RoboDK station: Sheet C - Bottom.rdk

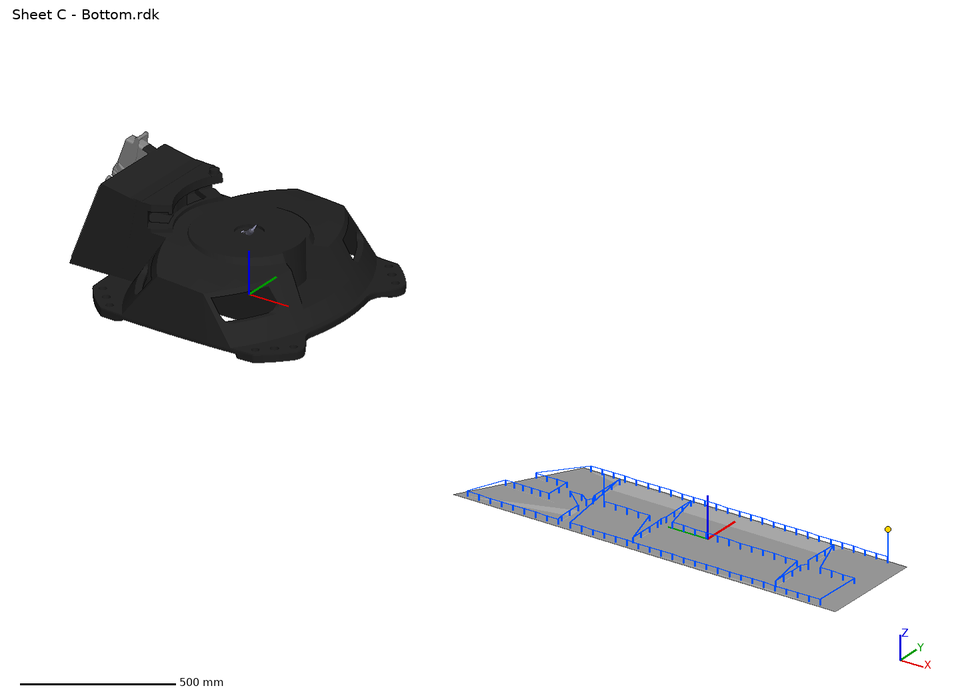
[picture v0: the station drawn from its stored meshes, robots at their saved joint values, targets as dots, program paths as lines]
Station Sheet C - Bottom (saved by RoboDK 5.2.3). Poses are relative to the parent item; angles as X-Y-Z fixed-axis rotations.
  - frame KUKA KR 210 R2700 extra Base at (0, 0, 0) mm
    - robot KUKA KR 210 R2700 extra: 6 axes, payload 210 kg, reach 2696 mm, repeatability 0.06 mm, weight 1068 kg
        joint limits [-185, -140, -120, -350, -125, -350] to [185, -5, 155, 350, 125, 350]; home [0, -90, 90, 0, 0, 0]; saved at [0.009, -34.349, 130.969, 180.008, 45.62, -179.999]
      - tool Spindle, TCP at (32, 0, 260) mm, rotated rx 0 ry 39 rz 0 deg, size 157.3 x 72 x 259.9 mm
  - frame Frame 2 at (1800, 0, -372.68) mm, rotated rx 0 ry 0 rz 90 deg
    - object Box 1 - Sheet C -  Bottom at (0, 0, 0) mm, size 400 x 1500 x 0.8 mm, geometry from Box 1 - Sheet C -  Bottom.stl
    - object Sheet C-box 1 Hole positioning Bottom at (0, 0, 0) mm, 120 curves, geometry from Point 120
  - machining project Path1 settings: rotZ(0) | rotX(0)*rotY(0) | rotz(0) | onStart | onPathStart | onApproach | onPoint | onRetract | onFinish | SetRPM(%1) | SetTool(%1) | Extruder(%1) | default | default | OutOnMov(%1) | OutOffMov(%1) | onPathFinish | M_RunCode(%1)
  - program Path1 (611 instructions, listed below)
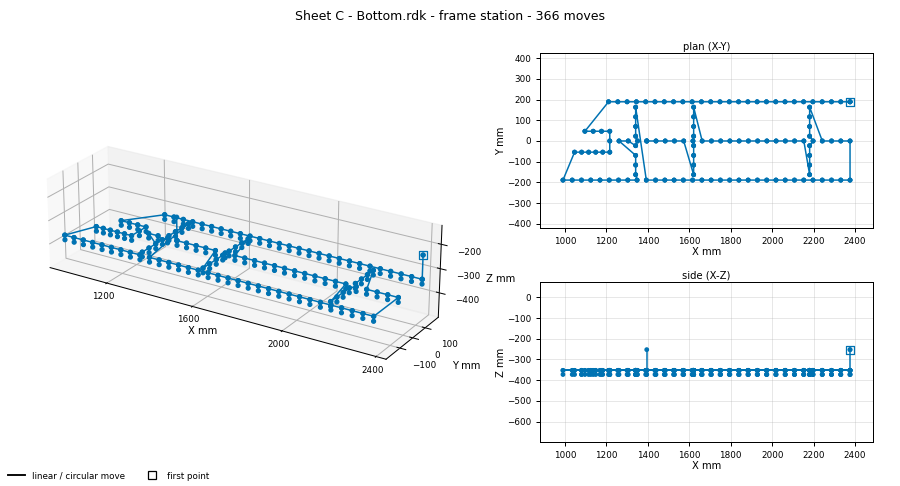
[picture p0: tool path of Sheet C - Bottom.rdk in frame station, 366 of 366 moves have a stored position in this frame; points joined in program order, loops and branches not executed]

--- program Path1 (robot KUKA KR 210 R2700 extra) ---
  Smooth(1)
  Set speed (1000.0 mm/s)
  Set Ref.: Frame 2
  Set Tool: Spindle
  Show Spindle
  MoveJ 1 to (189, -575.99, 120) mm, rotated rx -180 ry 0 rz 90 deg; joints [-5.138, -22.439, 74.968, 113.656, 3.528, -117.694]
  MoveL 2 to (189, -575.99, 120) mm, rotated rx -180 ry 0 rz 90 deg; joints [-5.138, -22.439, 74.968, 113.656, 3.528, -117.694]
  MoveL 3 to (189, -575.99, 20) mm, rotated rx 180 ry 0 rz 90 deg; joints [-5.138, -18.208, 72.448, 134.025, 4.496, -138.111]
  MoveL 4 to (189, -575.99, 20) mm, rotated rx 180 ry 0 rz 90 deg; joints [-5.138, -18.208, 72.448, 134.025, 4.496, -138.111]
  Set speed (50.0 mm/s)
  MoveL 5 to (189, -575.99, 0) mm, rotated rx -180 ry 0 rz 90 deg; joints [-5.138, -17.345, 71.889, 136.67, 4.711, -140.764]
  MoveL 6 to (189, -575.99, 20) mm, rotated rx 180 ry 0 rz 90 deg; joints [-5.138, -18.208, 72.448, 134.025, 4.496, -138.111]
  Set speed (1000.0 mm/s)
  MoveL 7 to (189, -531.14, 20) mm, rotated rx -180 ry 0 rz 90 deg; joints [-5.249, -19.449, 75.768, 147.536, 6.158, -151.77]
  Set speed (50.0 mm/s)
  MoveL 8 to (189, -531.14, 0) mm, rotated rx 180 ry 0 rz 90 deg; joints [-5.249, -18.579, 75.216, 149.054, 6.429, -153.297]
  MoveL 9 to (189, -531.14, 20) mm, rotated rx -180 ry 0 rz 90 deg; joints [-5.249, -19.449, 75.768, 147.536, 6.158, -151.77]
  Set speed (1000.0 mm/s)
  MoveL 10 to (189, -486.3, 20) mm, rotated rx 180 ry 0 rz 90 deg; joints [-5.366, -20.604, 78.961, 154.91, 7.977, -159.298]
  Set speed (50.0 mm/s)
  MoveL 11 to (189, -486.3, 0) mm, rotated rx -180 ry 0 rz 90 deg; joints [-5.366, -19.726, 78.415, 155.882, 8.281, -160.28]
  MoveL 12 to (189, -486.3, 20) mm, rotated rx 180 ry 0 rz 90 deg; joints [-5.366, -20.604, 78.961, 154.91, 7.977, -159.298]
  Set speed (1000.0 mm/s)
  MoveL 13 to (189, -441.45, 20) mm, rotated rx -180 ry 0 rz 90 deg; joints [-5.487, -21.682, 82.042, 159.405, 9.85, -163.953]
  Set speed (50.0 mm/s)
  MoveL 14 to (189, -441.45, 0) mm, rotated rx 180 ry 0 rz 90 deg; joints [-5.487, -20.792, 81.501, 160.086, 10.177, -164.645]
  MoveL 15 to (189, -441.45, 20) mm, rotated rx -180 ry 0 rz 90 deg; joints [-5.487, -21.682, 82.042, 159.405, 9.85, -163.953]
  Set speed (1000.0 mm/s)
  MoveL 16 to (189, -396.61, 20) mm, rotated rx 180 ry 0 rz 90 deg; joints [-5.615, -22.684, 85.023, 162.387, 11.74, -167.102]
  Set speed (50.0 mm/s)
  MoveL 17 to (189, -396.61, 0) mm, rotated rx 180 ry 0 rz 90 deg; joints [-5.615, -21.783, 84.484, 162.898, 12.086, -167.625]
  MoveL 18 to (189, -396.61, 20) mm, rotated rx 180 ry 0 rz 90 deg; joints [-5.615, -22.684, 85.023, 162.387, 11.74, -167.102]
  Set speed (1000.0 mm/s)
  MoveL 19 to (189, -351.76, 20) mm, rotated rx 180 ry 0 rz 90 deg; joints [-5.748, -23.614, 87.912, 164.494, 13.636, -169.383]
  Set speed (50.0 mm/s)
  MoveL 20 to (189, -351.76, 0) mm, rotated rx -180 ry 0 rz 90 deg; joints [-5.748, -22.7, 87.374, 164.896, 13.998, -169.798]
  MoveL 21 to (189, -351.76, 20) mm, rotated rx 180 ry 0 rz 90 deg; joints [-5.748, -23.614, 87.912, 164.494, 13.636, -169.383]
  Set speed (1000.0 mm/s)
  MoveL 22 to (189, -306.91, 20) mm, rotated rx 180 ry 0 rz 90 deg; joints [-5.887, -24.475, 90.718, 166.05, 15.532, -171.123]
  Set speed (50.0 mm/s)
  MoveL 23 to (189, -306.91, 0) mm, rotated rx 180 ry 0 rz 90 deg; joints [-5.887, -23.547, 90.179, 166.379, 15.909, -171.464]
  MoveL 24 to (189, -306.91, 20) mm, rotated rx 180 ry 0 rz 90 deg; joints [-5.887, -24.475, 90.718, 166.05, 15.532, -171.123]
  Set speed (1000.0 mm/s)
  MoveL 25 to (189, -262.07, 20) mm, rotated rx 180 ry 0 rz 90 deg; joints [-6.034, -25.267, 93.445, 167.24, 17.428, -172.504]
  Set speed (50.0 mm/s)
  MoveL 26 to (189, -262.07, 0) mm, rotated rx 180 ry 0 rz 90 deg; joints [-6.034, -24.325, 92.905, 167.516, 17.821, -172.794]
  MoveL 27 to (189, -262.07, 20) mm, rotated rx 180 ry 0 rz 90 deg; joints [-6.034, -25.267, 93.445, 167.24, 17.428, -172.504]
  Set speed (1000.0 mm/s)
  MoveL 28 to (189, -217.22, 20) mm, rotated rx 180 ry 0 rz 90 deg; joints [-6.188, -25.991, 96.102, 168.173, 19.328, -173.639]
  Set speed (50.0 mm/s)
  MoveL 29 to (189, -217.22, 0) mm, rotated rx 180 ry 0 rz 90 deg; joints [-6.188, -25.033, 95.559, 168.41, 19.734, -173.891]
  MoveL 30 to (189, -217.22, 20) mm, rotated rx 180 ry 0 rz 90 deg; joints [-6.188, -25.991, 96.102, 168.173, 19.328, -173.639]
  Set speed (1000.0 mm/s)
  MoveL 31 to (189, -172.37, 20) mm, rotated rx -180 ry 0 rz 90 deg; joints [-6.35, -26.648, 98.692, 168.919, 21.233, -174.597]
  Set speed (50.0 mm/s)
  MoveL 32 to (189, -172.37, 0) mm, rotated rx -180 ry 0 rz 90 deg; joints [-6.35, -25.673, 98.145, 169.126, 21.652, -174.82]
  MoveL 33 to (189, -172.37, 20) mm, rotated rx -180 ry 0 rz 90 deg; joints [-6.35, -26.648, 98.692, 168.919, 21.233, -174.597]
  Set speed (1000.0 mm/s)
  MoveL 34 to (189, -127.53, 20) mm, rotated rx -180 ry 0 rz 90 deg; joints [-6.521, -27.237, 101.217, 169.524, 23.145, -175.427]
  Set speed (50.0 mm/s)
  MoveL 35 to (189, -127.53, 0) mm, rotated rx -180 ry 0 rz 90 deg; joints [-6.521, -26.244, 100.665, 169.708, 23.578, -175.627]
  MoveL 36 to (189, -127.53, 20) mm, rotated rx -180 ry 0 rz 90 deg; joints [-6.521, -27.237, 101.217, 169.524, 23.145, -175.427]
  Set speed (1000.0 mm/s)
  MoveL 37 to (189, -82.68, 20) mm, rotated rx 180 ry 0 rz 90 deg; joints [-6.701, -27.756, 103.683, 170.02, 25.07, -176.161]
  Set speed (50.0 mm/s)
  MoveL 38 to (189, -82.68, 0) mm, rotated rx 180 ry 0 rz 90 deg; joints [-6.701, -26.744, 103.125, 170.184, 25.516, -176.343]
  MoveL 39 to (189, -82.68, 20) mm, rotated rx 180 ry 0 rz 90 deg; joints [-6.701, -27.756, 103.683, 170.02, 25.07, -176.161]
  Set speed (1000.0 mm/s)
  MoveL 40 to (189, -37.84, 20) mm, rotated rx -180 ry 0 rz 90 deg; joints [-6.891, -28.203, 106.092, 170.429, 27.009, -176.822]
  Set speed (50.0 mm/s)
  MoveL 41 to (189, -37.84, 0) mm, rotated rx -180 ry 0 rz 90 deg; joints [-6.891, -27.173, 105.527, 170.578, 27.468, -176.99]
  MoveL 42 to (189, -37.84, 20) mm, rotated rx -180 ry 0 rz 90 deg; joints [-6.891, -28.203, 106.092, 170.429, 27.009, -176.822]
  Set speed (1000.0 mm/s)
  MoveL 43 to (189, 7.01, 20) mm, rotated rx 180 ry 0 rz 90 deg; joints [-7.093, -28.577, 108.445, 170.767, 28.968, -177.429]
  Set speed (50.0 mm/s)
  MoveL 44 to (189, 7.01, 0) mm, rotated rx -180 ry 0 rz 90 deg; joints [-7.093, -27.526, 107.872, 170.903, 29.44, -177.585]
  MoveL 45 to (189, 7.01, 20) mm, rotated rx 180 ry 0 rz 90 deg; joints [-7.093, -28.577, 108.445, 170.767, 28.968, -177.429]
  Set speed (1000.0 mm/s)
  MoveL 46 to (189, 51.86, 20) mm, rotated rx -180 ry 0 rz 90 deg; joints [-7.306, -28.875, 110.745, 171.047, 30.95, -177.996]
  Set speed (50.0 mm/s)
  MoveL 47 to (189, 51.86, 0) mm, rotated rx 180 ry 0 rz 90 deg; joints [-7.306, -27.803, 110.163, 171.172, 31.434, -178.142]
  MoveL 48 to (189, 51.86, 20) mm, rotated rx -180 ry 0 rz 90 deg; joints [-7.306, -28.875, 110.745, 171.047, 30.95, -177.996]
  Set speed (1000.0 mm/s)
  MoveL 49 to (189, 96.7, 20) mm, rotated rx 180 ry 0 rz 90 deg; joints [-7.533, -29.093, 112.992, 171.278, 32.96, -178.532]
  Set speed (50.0 mm/s)
  MoveL 50 to (189, 96.7, 0) mm, rotated rx 180 ry 0 rz 90 deg; joints [-7.533, -27.999, 112.4, 171.393, 33.456, -178.67]
  MoveL 51 to (189, 96.7, 20) mm, rotated rx 180 ry 0 rz 90 deg; joints [-7.533, -29.093, 112.992, 171.278, 32.96, -178.532]
  Set speed (1000.0 mm/s)
  MoveL 52 to (189, 141.55, 20) mm, rotated rx 180 ry 0 rz 90 deg; joints [-7.774, -29.227, 115.187, 171.465, 35.001, -179.048]
  Set speed (50.0 mm/s)
  MoveL 53 to (189, 141.55, 0) mm, rotated rx -180 ry 0 rz 90 deg; joints [-7.774, -28.111, 114.584, 171.572, 35.509, -179.179]
  MoveL 54 to (189, 141.55, 20) mm, rotated rx 180 ry 0 rz 90 deg; joints [-7.774, -29.227, 115.187, 171.465, 35.001, -179.048]
  Set speed (1000.0 mm/s)
  MoveL 55 to (189, 186.39, 20) mm, rotated rx -180 ry 0 rz 90 deg; joints [-8.031, -29.272, 117.331, 171.615, 37.079, -179.55]
  Set speed (50.0 mm/s)
  MoveL 56 to (189, 186.39, 0) mm, rotated rx 180 ry 0 rz 90 deg; joints [-8.031, -28.133, 116.716, 171.714, 37.597, -179.676]
  MoveL 57 to (189, 186.39, 20) mm, rotated rx -180 ry 0 rz 90 deg; joints [-8.031, -29.272, 117.331, 171.615, 37.079, -179.55]
  Set speed (1000.0 mm/s)
  MoveL 58 to (189, 231.24, 20) mm, rotated rx -180 ry 0 rz 90 deg; joints [-8.305, -29.223, 119.424, 171.73, 39.199, -180.046]
  Set speed (50.0 mm/s)
  MoveL 59 to (189, 231.24, 0) mm, rotated rx 180 ry 0 rz 90 deg; joints [-8.305, -28.061, 118.796, 171.823, 39.727, -180.166]
  MoveL 60 to (189, 231.24, 20) mm, rotated rx -180 ry 0 rz 90 deg; joints [-8.305, -29.223, 119.424, 171.73, 39.199, -180.046]
  Set speed (1000.0 mm/s)
  MoveL 61 to (189, 276.09, 20) mm, rotated rx -180 ry 0 rz 90 deg; joints [-8.599, -29.075, 121.466, 171.814, 41.365, -180.541]
  Set speed (50.0 mm/s)
  MoveL 62 to (189, 276.09, 0) mm, rotated rx -180 ry 0 rz 90 deg; joints [-8.599, -27.889, 120.823, 171.901, 41.903, -180.657]
  MoveL 63 to (189, 276.09, 20) mm, rotated rx -180 ry 0 rz 90 deg; joints [-8.599, -29.075, 121.466, 171.814, 41.365, -180.541]
  Set speed (1000.0 mm/s)
  MoveL 64 to (189, 320.93, 20) mm, rotated rx 180 ry 0 rz 90 deg; joints [-8.914, -28.82, 123.454, 171.868, 43.583, -181.04]
  Set speed (50.0 mm/s)
  MoveL 65 to (189, 320.93, 0) mm, rotated rx -180 ry 0 rz 90 deg; joints [-8.914, -27.611, 122.796, 171.949, 44.129, -181.153]
  MoveL 66 to (189, 320.93, 20) mm, rotated rx 180 ry 0 rz 90 deg; joints [-8.914, -28.82, 123.454, 171.868, 43.583, -181.04]
  Set speed (1000.0 mm/s)
  MoveL 67 to (189, 365.78, 20) mm, rotated rx 180 ry 0 rz 90 deg; joints [-9.253, -28.451, 125.389, 171.894, 45.859, -181.551]
  Set speed (50.0 mm/s)
  MoveL 68 to (189, 365.78, 0) mm, rotated rx -180 ry 0 rz 90 deg; joints [-9.253, -27.219, 124.715, 171.969, 46.412, -181.66]
  MoveL 69 to (189, 365.78, 20) mm, rotated rx 180 ry 0 rz 90 deg; joints [-9.253, -28.451, 125.389, 171.894, 45.859, -181.551]
  Set speed (1000.0 mm/s)
  MoveL 70 to (189, 410.63, 20) mm, rotated rx 180 ry 0 rz 90 deg; joints [-9.618, -27.959, 127.268, 171.892, 48.199, -182.078]
  Set speed (50.0 mm/s)
  MoveL 71 to (189, 410.63, 0) mm, rotated rx 180 ry 0 rz 90 deg; joints [-9.618, -26.705, 126.576, 171.962, 48.756, -182.183]
  MoveL 72 to (189, 410.63, 20) mm, rotated rx 180 ry 0 rz 90 deg; joints [-9.618, -27.959, 127.268, 171.892, 48.199, -182.078]
  Set speed (1000.0 mm/s)
  MoveL 73 to (189, 455.47, 20) mm, rotated rx -180 ry 0 rz 90 deg; joints [-10.013, -27.337, 129.088, 171.86, 50.607, -182.626]
  Set speed (50.0 mm/s)
  MoveL 74 to (189, 455.47, 0) mm, rotated rx 180 ry 0 rz 90 deg; joints [-10.013, -26.061, 128.379, 171.925, 51.167, -182.729]
  MoveL 75 to (189, 455.47, 20) mm, rotated rx -180 ry 0 rz 90 deg; joints [-10.013, -27.337, 129.088, 171.86, 50.607, -182.626]
  Set speed (1000.0 mm/s)
  MoveL 76 to (189, 500.32, 20) mm, rotated rx -180 ry 0 rz 90 deg; joints [-10.441, -26.573, 130.848, 171.8, 53.091, -183.204]
  Set speed (50.0 mm/s)
  MoveL 77 to (189, 500.32, 0) mm, rotated rx 180 ry 0 rz 90 deg; joints [-10.441, -25.278, 130.119, 171.859, 53.651, -183.304]
  MoveL 78 to (189, 500.32, 20) mm, rotated rx -180 ry 0 rz 90 deg; joints [-10.441, -26.573, 130.848, 171.8, 53.091, -183.204]
  Set speed (1000.0 mm/s)
  MoveL 79 to (189, 545.16, 20) mm, rotated rx 180 ry 0 rz 90 deg; joints [-10.907, -25.659, 132.544, 171.708, 55.656, -183.817]
  Set speed (50.0 mm/s)
  MoveL 80 to (189, 545.16, 0) mm, rotated rx -180 ry 0 rz 90 deg; joints [-10.907, -24.347, 131.794, 171.762, 56.212, -183.914]
  MoveL 81 to (189, 545.16, 20) mm, rotated rx 180 ry 0 rz 90 deg; joints [-10.907, -25.659, 132.544, 171.708, 55.656, -183.817]
  Set speed (1000.0 mm/s)
  MoveL 82 to (189, 590.01, 20) mm, rotated rx 180 ry 0 rz 90 deg; joints [-11.417, -24.583, 134.171, 171.582, 58.308, -184.473]
  Set speed (50.0 mm/s)
  MoveL 83 to (189, 590.01, 0) mm, rotated rx 180 ry 0 rz 90 deg; joints [-11.417, -23.257, 133.4, 171.631, 58.856, -184.568]
  MoveL 84 to (189, 590.01, 20) mm, rotated rx 180 ry 0 rz 90 deg; joints [-11.417, -24.583, 134.171, 171.582, 58.308, -184.473]
  Set speed (1000.0 mm/s)
  MoveL 85 to (46.83, 704.01, 20) mm, rotated rx -180 ry 0 rz 90 deg; joints [-3.261, -20.272, 138.599, 177.776, 67.298, -181.677]
  Set speed (50.0 mm/s)
  MoveL 86 to (46.83, 704.01, 0) mm, rotated rx -180 ry 0 rz 90 deg; joints [-3.261, -18.933, 137.76, 177.784, 67.797, -181.698]
  MoveL 87 to (46.83, 704.01, 20) mm, rotated rx -180 ry 0 rz 90 deg; joints [-3.261, -20.272, 138.599, 177.776, 67.298, -181.677]
  Set speed (1000.0 mm/s)
  MoveL 88 to (46.83, 664.01, 20) mm, rotated rx -180 ry 0 rz 90 deg; joints [-3.11, -21.766, 137.33, 177.833, 64.539, -181.486]
  Set speed (50.0 mm/s)
  MoveL 89 to (46.83, 664.01, 0) mm, rotated rx 180 ry 0 rz 90 deg; joints [-3.11, -20.425, 136.512, 177.842, 65.061, -181.508]
  MoveL 90 to (46.83, 664.01, 20) mm, rotated rx -180 ry 0 rz 90 deg; joints [-3.11, -21.766, 137.33, 177.833, 64.539, -181.486]
  Set speed (1000.0 mm/s)
  MoveL 91 to (46.83, 624.01, 20) mm, rotated rx -180 ry 0 rz 90 deg; joints [-2.972, -23.094, 135.993, 177.88, 61.877, -181.311]
  Set speed (50.0 mm/s)
  MoveL 92 to (46.83, 624.01, 0) mm, rotated rx -180 ry 0 rz 90 deg; joints [-2.972, -21.757, 135.196, 177.89, 62.416, -181.333]
  MoveL 93 to (46.83, 624.01, 20) mm, rotated rx -180 ry 0 rz 90 deg; joints [-2.972, -23.094, 135.993, 177.88, 61.877, -181.311]
  Set speed (1000.0 mm/s)
  MoveL 94 to (46.83, 584.01, 20) mm, rotated rx -180 ry 0 rz 90 deg; joints [-2.846, -24.267, 134.593, 177.917, 59.309, -181.149]
  Set speed (50.0 mm/s)
  MoveL 95 to (46.83, 584.01, 0) mm, rotated rx 180 ry 0 rz 90 deg; joints [-2.846, -22.938, 133.816, 177.929, 59.86, -181.173]
  MoveL 96 to (46.83, 584.01, 20) mm, rotated rx -180 ry 0 rz 90 deg; joints [-2.846, -24.267, 134.593, 177.917, 59.309, -181.149]
  Set speed (1000.0 mm/s)
  MoveL 97 to (-0.17, 584.01, 20) mm, rotated rx -180 ry 0 rz 90 deg; joints [0.01, -24.235, 134.635, 180.008, 59.4, -179.996]
  Set speed (50.0 mm/s)
  MoveL 98 to (-0.17, 584.01, 0) mm, rotated rx -180 ry 0 rz 90 deg; joints [0.01, -22.906, 133.857, 180.008, 59.952, -179.996]
  MoveL 99 to (-0.17, 584.01, 20) mm, rotated rx -180 ry 0 rz 90 deg; joints [0.01, -24.235, 134.635, 180.008, 59.4, -179.996]
  Set speed (1000.0 mm/s)
  MoveL 100 to (-54.17, 584.01, 20) mm, rotated rx -180 ry 0 rz 90 deg; joints [3.291, -24.277, 134.579, 182.409, 59.278, -178.672]
  Set speed (50.0 mm/s)
  MoveL 101 to (-54.17, 584.01, 0) mm, rotated rx 180 ry 0 rz 90 deg; joints [3.291, -22.949, 133.803, 182.395, 59.829, -178.645]
  MoveL 102 to (-54.17, 584.01, 20) mm, rotated rx -180 ry 0 rz 90 deg; joints [3.291, -24.277, 134.579, 182.409, 59.278, -178.672]
  Set speed (1000.0 mm/s)
  MoveL 103 to (-54.17, 618.01, 20) mm, rotated rx -180 ry 0 rz 90 deg; joints [3.414, -23.292, 135.773, 182.445, 61.453, -178.514]
  Set speed (50.0 mm/s)
  MoveL 104 to (-54.17, 618.01, 0) mm, rotated rx 180 ry 0 rz 90 deg; joints [3.414, -21.957, 134.979, 182.433, 61.994, -178.488]
  MoveL 105 to (-54.17, 618.01, 20) mm, rotated rx -180 ry 0 rz 90 deg; joints [3.414, -23.292, 135.773, 182.445, 61.453, -178.514]
  Set speed (1000.0 mm/s)
  MoveL 106 to (-54.17, 652.01, 20) mm, rotated rx -180 ry 0 rz 90 deg; joints [3.547, -22.196, 136.922, 182.489, 63.694, -178.346]
  Set speed (50.0 mm/s)
  MoveL 107 to (-54.17, 652.01, 0) mm, rotated rx -180 ry 0 rz 90 deg; joints [3.547, -20.856, 136.11, 182.478, 64.221, -178.32]
  MoveL 108 to (-54.17, 652.01, 20) mm, rotated rx -180 ry 0 rz 90 deg; joints [3.547, -22.196, 136.922, 182.489, 63.694, -178.346]
  Set speed (1000.0 mm/s)
  MoveL 109 to (-54.17, 686.01, 20) mm, rotated rx -180 ry 0 rz 90 deg; joints [3.69, -20.982, 138.023, 182.541, 66.004, -178.165]
  Set speed (50.0 mm/s)
  MoveL 110 to (-54.17, 686.01, 0) mm, rotated rx -180 ry 0 rz 90 deg; joints [3.69, -19.641, 137.193, 182.531, 66.514, -178.14]
  MoveL 111 to (-54.17, 686.01, 20) mm, rotated rx -180 ry 0 rz 90 deg; joints [3.69, -20.982, 138.023, 182.541, 66.004, -178.165]
  Set speed (1000.0 mm/s)
  MoveL 112 to (-54.17, 720.01, 20) mm, rotated rx -180 ry 0 rz 90 deg; joints [3.845, -19.645, 139.073, 182.602, 68.386, -177.969]
  Set speed (50.0 mm/s)
  MoveL 113 to (-54.17, 720.01, 0) mm, rotated rx 180 ry 0 rz 90 deg; joints [3.845, -18.308, 138.226, 182.593, 68.874, -177.945]
  MoveL 114 to (-54.17, 720.01, 20) mm, rotated rx -180 ry 0 rz 90 deg; joints [3.845, -19.645, 139.073, 182.602, 68.386, -177.969]
  Set speed (1000.0 mm/s)
  MoveL 115 to (-54.17, 754.01, 20) mm, rotated rx 180 ry 0 rz 90 deg; joints [4.014, -18.181, 140.071, 182.673, 70.84, -177.756]
  Set speed (50.0 mm/s)
  MoveL 116 to (-54.17, 754.01, 0) mm, rotated rx -180 ry 0 rz 90 deg; joints [4.014, -16.852, 139.205, 182.666, 71.302, -177.734]
  MoveL 117 to (-54.17, 754.01, 20) mm, rotated rx 180 ry 0 rz 90 deg; joints [4.014, -18.181, 140.071, 182.673, 70.84, -177.756]
  Set speed (1000.0 mm/s)
  MoveL 118 to (-189, 810.01, 20) mm, rotated rx 180 ry 0 rz 90 deg; joints [14.788, -16.611, 140.997, 189.687, 72.681, -171.315]
  Set speed (50.0 mm/s)
  MoveL 119 to (-189, 810.01, 0) mm, rotated rx 180 ry 0 rz 90 deg; joints [14.788, -15.296, 140.112, 189.664, 73.105, -171.239]
  MoveL 120 to (-189, 810.01, 20) mm, rotated rx 180 ry 0 rz 90 deg; joints [14.788, -16.611, 140.997, 189.687, 72.681, -171.315]
  Set speed (1000.0 mm/s)
  MoveL 121 to (-189, 765.3, 20) mm, rotated rx -180 ry 0 rz 90 deg; joints [13.954, -18.623, 139.784, 189.319, 69.574, -172.348]
  Set speed (50.0 mm/s)
  MoveL 122 to (-189, 765.3, 0) mm, rotated rx -180 ry 0 rz 90 deg; joints [13.954, -17.292, 138.923, 189.291, 70.039, -172.267]
  MoveL 123 to (-189, 765.3, 20) mm, rotated rx -180 ry 0 rz 90 deg; joints [13.954, -18.623, 139.784, 189.319, 69.574, -172.348]
  Set speed (1000.0 mm/s)
  MoveL 124 to (-189, 720.59, 20) mm, rotated rx 180 ry 0 rz 90 deg; joints [13.207, -20.428, 138.476, 189.016, 66.561, -173.276]
  Set speed (50.0 mm/s)
  MoveL 125 to (-189, 720.59, 0) mm, rotated rx -180 ry 0 rz 90 deg; joints [13.207, -19.088, 137.639, 188.983, 67.057, -173.19]
  MoveL 126 to (-189, 720.59, 20) mm, rotated rx 180 ry 0 rz 90 deg; joints [13.207, -20.428, 138.476, 189.016, 66.561, -173.276]
  Set speed (1000.0 mm/s)
  MoveL 127 to (-189, 675.88, 20) mm, rotated rx -180 ry 0 rz 90 deg; joints [12.535, -22.031, 137.08, 188.768, 63.643, -174.114]
  Set speed (50.0 mm/s)
  MoveL 128 to (-189, 675.88, 0) mm, rotated rx 180 ry 0 rz 90 deg; joints [12.535, -20.691, 136.266, 188.729, 64.163, -174.025]
  MoveL 129 to (-189, 675.88, 20) mm, rotated rx -180 ry 0 rz 90 deg; joints [12.535, -22.031, 137.08, 188.768, 63.643, -174.114]
  Set speed (1000.0 mm/s)
  MoveL 130 to (-189, 631.17, 20) mm, rotated rx 180 ry 0 rz 90 deg; joints [11.927, -23.443, 135.601, 188.567, 60.822, -174.878]
  Set speed (50.0 mm/s)
  MoveL 131 to (-189, 631.17, 0) mm, rotated rx -180 ry 0 rz 90 deg; joints [11.927, -22.109, 134.809, 188.522, 61.359, -174.786]
  MoveL 132 to (-189, 631.17, 20) mm, rotated rx 180 ry 0 rz 90 deg; joints [11.927, -23.443, 135.601, 188.567, 60.822, -174.878]
  Set speed (1000.0 mm/s)
  MoveL 133 to (-189, 586.46, 20) mm, rotated rx -180 ry 0 rz 90 deg; joints [11.375, -24.674, 134.045, 188.407, 58.095, -175.581]
  Set speed (50.0 mm/s)
  MoveL 134 to (-189, 586.46, 0) mm, rotated rx -180 ry 0 rz 90 deg; joints [11.375, -23.349, 133.276, 188.357, 58.644, -175.485]
  MoveL 135 to (-189, 586.46, 20) mm, rotated rx -180 ry 0 rz 90 deg; joints [11.375, -24.674, 134.045, 188.407, 58.095, -175.581]
  Set speed (1000.0 mm/s)
  MoveL 136 to (-189, 541.75, 20) mm, rotated rx -180 ry 0 rz 90 deg; joints [10.871, -25.734, 132.417, 188.284, 55.458, -176.231]
  Set speed (50.0 mm/s)
  MoveL 137 to (-189, 541.75, 0) mm, rotated rx -180 ry 0 rz 90 deg; joints [10.871, -24.423, 131.669, 188.229, 56.015, -176.134]
  MoveL 138 to (-189, 541.75, 20) mm, rotated rx -180 ry 0 rz 90 deg; joints [10.871, -25.734, 132.417, 188.284, 55.458, -176.231]
  Set speed (1000.0 mm/s)
  MoveL 139 to (-189, 497.04, 20) mm, rotated rx -180 ry 0 rz 90 deg; joints [10.409, -26.634, 130.722, 188.195, 52.907, -176.84]
  Set speed (50.0 mm/s)
  MoveL 140 to (-189, 497.04, 0) mm, rotated rx -180 ry 0 rz 90 deg; joints [10.409, -25.341, 129.994, 188.135, 53.467, -176.739]
  MoveL 141 to (-189, 497.04, 20) mm, rotated rx -180 ry 0 rz 90 deg; joints [10.409, -26.634, 130.722, 188.195, 52.907, -176.84]
  Set speed (1000.0 mm/s)
  MoveL 142 to (-189, 452.33, 20) mm, rotated rx 180 ry 0 rz 90 deg; joints [9.984, -27.385, 128.963, 188.136, 50.436, -177.413]
  Set speed (50.0 mm/s)
  MoveL 143 to (-189, 452.33, 0) mm, rotated rx -180 ry 0 rz 90 deg; joints [9.984, -26.111, 128.254, 188.071, 50.996, -177.31]
  MoveL 144 to (-189, 452.33, 20) mm, rotated rx 180 ry 0 rz 90 deg; joints [9.984, -27.385, 128.963, 188.136, 50.436, -177.413]
  Set speed (1000.0 mm/s)
  MoveL 145 to (-163, 459.01, 20) mm, rotated rx 180 ry 0 rz 90 deg; joints [8.686, -27.214, 129.4, 187.017, 51.075, -177.651]
  Set speed (50.0 mm/s)
  MoveL 146 to (-163, 459.01, 0) mm, rotated rx -180 ry 0 rz 90 deg; joints [8.686, -25.935, 128.687, 186.962, 51.636, -177.563]
  MoveL 147 to (-163, 459.01, 20) mm, rotated rx 180 ry 0 rz 90 deg; joints [8.686, -27.214, 129.4, 187.017, 51.075, -177.651]
  Set speed (1000.0 mm/s)
  MoveL 148 to (-116.33, 459.01, 20) mm, rotated rx 180 ry 0 rz 90 deg; joints [6.223, -27.114, 129.644, 185.002, 51.471, -178.277]
  Set speed (50.0 mm/s)
  MoveL 149 to (-116.33, 459.01, 0) mm, rotated rx 180 ry 0 rz 90 deg; joints [6.223, -25.832, 128.928, 184.964, 52.035, -178.215]
  MoveL 150 to (-116.33, 459.01, 20) mm, rotated rx 180 ry 0 rz 90 deg; joints [6.223, -27.114, 129.644, 185.002, 51.471, -178.277]
  Set speed (1000.0 mm/s)
  MoveL 151 to (-69.67, 459.01, 20) mm, rotated rx -180 ry 0 rz 90 deg; joints [3.736, -27.046, 129.806, 182.994, 51.739, -178.95]
  Set speed (50.0 mm/s)
  MoveL 152 to (-69.67, 459.01, 0) mm, rotated rx 180 ry 0 rz 90 deg; joints [3.736, -25.763, 129.089, 182.971, 52.304, -178.912]
  MoveL 153 to (-69.67, 459.01, 20) mm, rotated rx -180 ry 0 rz 90 deg; joints [3.736, -27.046, 129.806, 182.994, 51.739, -178.95]
  Set speed (1000.0 mm/s)
  MoveL 154 to (-0.17, 539.39, 20) mm, rotated rx 180 ry 0 rz 90 deg; joints [0.01, -25.375, 133.004, 180.007, 56.629, -179.996]
  Set speed (50.0 mm/s)
  MoveL 155 to (-0.17, 539.39, 0) mm, rotated rx 180 ry 0 rz 90 deg; joints [0.01, -24.06, 132.249, 180.007, 57.189, -179.996]
  MoveL 156 to (-0.17, 539.39, 20) mm, rotated rx 180 ry 0 rz 90 deg; joints [0.01, -25.375, 133.004, 180.007, 56.629, -179.996]
  Set speed (1000.0 mm/s)
  MoveL 157 to (-0.17, 494.78, 20) mm, rotated rx 180 ry 0 rz 90 deg; joints [0.009, -26.345, 131.306, 180.007, 53.961, -179.997]
  Set speed (50.0 mm/s)
  MoveL 158 to (-0.17, 494.78, 0) mm, rotated rx -180 ry 0 rz 90 deg; joints [0.009, -25.046, 130.571, 180.007, 54.526, -179.997]
  MoveL 159 to (-0.17, 494.78, 20) mm, rotated rx 180 ry 0 rz 90 deg; joints [0.009, -26.345, 131.306, 180.007, 53.961, -179.997]
  Set speed (1000.0 mm/s)
  MoveL 160 to (-23, 459.01, 20) mm, rotated rx 180 ry 0 rz 90 deg; joints [1.235, -27.011, 129.887, 180.988, 51.873, -179.65]
  Set speed (50.0 mm/s)
  MoveL 161 to (-23, 459.01, 0) mm, rotated rx 180 ry 0 rz 90 deg; joints [1.235, -25.727, 129.169, 180.98, 52.439, -179.638]
  MoveL 162 to (-23, 459.01, 20) mm, rotated rx 180 ry 0 rz 90 deg; joints [1.235, -27.011, 129.887, 180.988, 51.873, -179.65]
  Set speed (1000.0 mm/s)
  MoveL 163 to (-0.17, 450.16, 20) mm, rotated rx 180 ry 0 rz 90 deg; joints [0.009, -27.156, 129.542, 180.007, 51.387, -179.998]
  Set speed (50.0 mm/s)
  MoveL 164 to (-0.17, 450.16, 0) mm, rotated rx -180 ry 0 rz 90 deg; joints [0.009, -25.876, 128.828, 180.007, 51.952, -179.997]
  MoveL 165 to (-0.17, 450.16, 20) mm, rotated rx 180 ry 0 rz 90 deg; joints [0.009, -27.156, 129.542, 180.007, 51.387, -179.998]
  Set speed (1000.0 mm/s)
  MoveL 166 to (23, 459.01, 20) mm, rotated rx -180 ry 0 rz 90 deg; joints [-1.235, -27.011, 129.887, 179.012, 51.873, -180.35]
  Set speed (50.0 mm/s)
  MoveL 167 to (23, 459.01, 0) mm, rotated rx -180 ry 0 rz 90 deg; joints [-1.235, -25.727, 129.169, 179.02, 52.439, -180.362]
  MoveL 168 to (23, 459.01, 20) mm, rotated rx -180 ry 0 rz 90 deg; joints [-1.235, -27.011, 129.887, 179.012, 51.873, -180.35]
  Set speed (1000.0 mm/s)
  MoveL 169 to (69.67, 459.01, 20) mm, rotated rx 180 ry 0 rz 90 deg; joints [-3.736, -27.046, 129.806, 177.006, 51.739, -181.05]
  Set speed (50.0 mm/s)
  MoveL 170 to (69.67, 459.01, 0) mm, rotated rx -180 ry 0 rz 90 deg; joints [-3.736, -25.763, 129.089, 177.029, 52.304, -181.088]
  MoveL 171 to (69.67, 459.01, 20) mm, rotated rx 180 ry 0 rz 90 deg; joints [-3.736, -27.046, 129.806, 177.006, 51.739, -181.05]
  Set speed (1000.0 mm/s)
  MoveL 172 to (116.33, 459.01, 20) mm, rotated rx -180 ry 0 rz 90 deg; joints [-6.223, -27.114, 129.644, 174.998, 51.471, -181.723]
  Set speed (50.0 mm/s)
  MoveL 173 to (116.33, 459.01, 0) mm, rotated rx 180 ry 0 rz 90 deg; joints [-6.223, -25.832, 128.928, 175.036, 52.035, -181.785]
  MoveL 174 to (116.33, 459.01, 20) mm, rotated rx -180 ry 0 rz 90 deg; joints [-6.223, -27.114, 129.644, 174.998, 51.471, -181.723]
  Set speed (1000.0 mm/s)
  MoveL 175 to (163, 459.01, 20) mm, rotated rx -180 ry 0 rz 90 deg; joints [-8.686, -27.214, 129.4, 172.983, 51.075, -182.349]
  Set speed (50.0 mm/s)
  MoveL 176 to (163, 459.01, 0) mm, rotated rx -180 ry 0 rz 90 deg; joints [-8.686, -25.935, 128.687, 173.038, 51.636, -182.437]
  MoveL 177 to (163, 459.01, 20) mm, rotated rx -180 ry 0 rz 90 deg; joints [-8.686, -27.214, 129.4, 172.983, 51.075, -182.349]
  Set speed (1000.0 mm/s)
  MoveL 178 to (-189, 407.62, 20) mm, rotated rx 180 ry 0 rz 90 deg; joints [9.593, -27.996, 127.143, 188.107, 48.04, -177.958]
  Set speed (50.0 mm/s)
  MoveL 179 to (-189, 407.62, 0) mm, rotated rx -180 ry 0 rz 90 deg; joints [9.593, -26.743, 126.453, 188.037, 48.597, -177.853]
  MoveL 180 to (-189, 407.62, 20) mm, rotated rx 180 ry 0 rz 90 deg; joints [9.593, -27.996, 127.143, 188.107, 48.04, -177.958]
  Set speed (1000.0 mm/s)
  MoveL 181 to (-189, 362.91, 20) mm, rotated rx -180 ry 0 rz 90 deg; joints [9.23, -28.478, 125.267, 188.107, 45.712, -178.482]
  Set speed (50.0 mm/s)
  MoveL 182 to (-189, 362.91, 0) mm, rotated rx -180 ry 0 rz 90 deg; joints [9.23, -27.247, 124.594, 188.031, 46.264, -178.373]
  MoveL 183 to (-189, 362.91, 20) mm, rotated rx -180 ry 0 rz 90 deg; joints [9.23, -28.478, 125.267, 188.107, 45.712, -178.482]
  Set speed (1000.0 mm/s)
  MoveL 184 to (-189, 318.2, 20) mm, rotated rx -180 ry 0 rz 90 deg; joints [8.894, -28.839, 123.334, 188.134, 43.447, -178.99]
  Set speed (50.0 mm/s)
  MoveL 185 to (-189, 318.2, 0) mm, rotated rx 180 ry 0 rz 90 deg; joints [8.894, -27.631, 122.678, 188.053, 43.992, -178.878]
  MoveL 186 to (-189, 318.2, 20) mm, rotated rx -180 ry 0 rz 90 deg; joints [8.894, -28.839, 123.334, 188.134, 43.447, -178.99]
  Set speed (1000.0 mm/s)
  MoveL 187 to (-189, 273.49, 20) mm, rotated rx -180 ry 0 rz 90 deg; joints [8.581, -29.086, 121.349, 188.19, 41.238, -179.488]
  Set speed (50.0 mm/s)
  MoveL 188 to (-189, 273.49, 0) mm, rotated rx 180 ry 0 rz 90 deg; joints [8.581, -27.902, 120.707, 188.103, 41.776, -179.372]
  MoveL 189 to (-189, 273.49, 20) mm, rotated rx -180 ry 0 rz 90 deg; joints [8.581, -29.086, 121.349, 188.19, 41.238, -179.488]
  Set speed (1000.0 mm/s)
  MoveL 190 to (-189, 228.78, 20) mm, rotated rx 180 ry 0 rz 90 deg; joints [8.29, -29.229, 119.311, 188.275, 39.081, -179.981]
  Set speed (50.0 mm/s)
  MoveL 191 to (-189, 228.78, 0) mm, rotated rx 180 ry 0 rz 90 deg; joints [8.29, -28.068, 118.683, 188.182, 39.609, -179.861]
  MoveL 192 to (-189, 228.78, 20) mm, rotated rx 180 ry 0 rz 90 deg; joints [8.29, -29.229, 119.311, 188.275, 39.081, -179.981]
  Set speed (1000.0 mm/s)
  MoveL 193 to (-189, 184.07, 20) mm, rotated rx 180 ry 0 rz 90 deg; joints [8.017, -29.272, 117.222, 188.392, 36.971, -180.475]
  Set speed (50.0 mm/s)
  MoveL 194 to (-189, 184.07, 0) mm, rotated rx 180 ry 0 rz 90 deg; joints [8.017, -28.134, 116.607, 188.292, 37.488, -180.35]
  MoveL 195 to (-189, 184.07, 20) mm, rotated rx 180 ry 0 rz 90 deg; joints [8.017, -29.272, 117.222, 188.392, 36.971, -180.475]
  Set speed (1000.0 mm/s)
  MoveL 196 to (-189, 139.36, 20) mm, rotated rx -180 ry 0 rz 90 deg; joints [7.762, -29.222, 115.081, 188.543, 34.901, -180.977]
  Set speed (50.0 mm/s)
  MoveL 197 to (-189, 139.36, 0) mm, rotated rx -180 ry 0 rz 90 deg; joints [7.762, -28.107, 114.479, 188.436, 35.408, -180.845]
  MoveL 198 to (-189, 139.36, 20) mm, rotated rx -180 ry 0 rz 90 deg; joints [7.762, -29.222, 115.081, 188.543, 34.901, -180.977]
  Set speed (1000.0 mm/s)
  MoveL 199 to (-189, 94.65, 20) mm, rotated rx -180 ry 0 rz 90 deg; joints [7.522, -29.085, 112.89, 188.732, 32.867, -181.492]
  Set speed (50.0 mm/s)
  MoveL 200 to (-189, 94.65, 0) mm, rotated rx 180 ry 0 rz 90 deg; joints [7.522, -27.992, 112.298, 188.616, 33.363, -181.353]
  MoveL 201 to (-189, 94.65, 20) mm, rotated rx -180 ry 0 rz 90 deg; joints [7.522, -29.085, 112.89, 188.732, 32.867, -181.492]
  Set speed (1000.0 mm/s)
  MoveL 202 to (-189, 49.95, 20) mm, rotated rx 180 ry 0 rz 90 deg; joints [7.297, -28.864, 110.648, 188.964, 30.865, -182.028]
  Set speed (50.0 mm/s)
  MoveL 203 to (-189, 49.95, 0) mm, rotated rx 180 ry 0 rz 90 deg; joints [7.297, -27.793, 110.066, 188.838, 31.349, -181.881]
  MoveL 204 to (-189, 49.95, 20) mm, rotated rx 180 ry 0 rz 90 deg; joints [7.297, -28.864, 110.648, 188.964, 30.865, -182.028]
  Set speed (1000.0 mm/s)
  MoveL 205 to (-189, 5.24, 20) mm, rotated rx -180 ry 0 rz 90 deg; joints [7.085, -28.564, 108.353, 189.245, 28.89, -182.594]
  Set speed (50.0 mm/s)
  MoveL 206 to (-189, 5.24, 0) mm, rotated rx -180 ry 0 rz 90 deg; joints [7.085, -27.514, 107.78, 189.108, 29.362, -182.437]
  MoveL 207 to (-189, 5.24, 20) mm, rotated rx -180 ry 0 rz 90 deg; joints [7.085, -28.564, 108.353, 189.245, 28.89, -182.594]
  Set speed (1000.0 mm/s)
  MoveL 208 to (-189, -39.47, 20) mm, rotated rx 180 ry 0 rz 90 deg; joints [6.884, -28.188, 106.005, 189.585, 26.938, -183.201]
  Set speed (50.0 mm/s)
  MoveL 209 to (-189, -39.47, 0) mm, rotated rx 180 ry 0 rz 90 deg; joints [6.884, -27.158, 105.44, 189.435, 27.397, -183.033]
  MoveL 210 to (-189, -39.47, 20) mm, rotated rx 180 ry 0 rz 90 deg; joints [6.884, -28.188, 106.005, 189.585, 26.938, -183.201]
  Set speed (1000.0 mm/s)
  MoveL 211 to (-189, -84.18, 20) mm, rotated rx -180 ry 0 rz 90 deg; joints [6.695, -27.739, 103.602, 189.995, 25.005, -183.863]
  Set speed (50.0 mm/s)
  MoveL 212 to (-189, -84.18, 0) mm, rotated rx 180 ry 0 rz 90 deg; joints [6.695, -26.729, 103.044, 189.83, 25.451, -183.68]
  MoveL 213 to (-189, -84.18, 20) mm, rotated rx -180 ry 0 rz 90 deg; joints [6.695, -27.739, 103.602, 189.995, 25.005, -183.863]
  Set speed (1000.0 mm/s)
  MoveL 214 to (-189, -128.89, 20) mm, rotated rx -180 ry 0 rz 90 deg; joints [6.516, -27.22, 101.142, 190.493, 23.087, -184.597]
  Set speed (50.0 mm/s)
  MoveL 215 to (-189, -128.89, 0) mm, rotated rx -180 ry 0 rz 90 deg; joints [6.516, -26.228, 100.59, 190.308, 23.52, -184.396]
  MoveL 216 to (-189, -128.89, 20) mm, rotated rx -180 ry 0 rz 90 deg; joints [6.516, -27.22, 101.142, 190.493, 23.087, -184.597]
  Set speed (1000.0 mm/s)
  MoveL 217 to (-189, -173.6, 20) mm, rotated rx -180 ry 0 rz 90 deg; joints [6.346, -26.631, 98.622, 191.1, 21.18, -185.427]
  Set speed (50.0 mm/s)
  MoveL 218 to (-189, -173.6, 0) mm, rotated rx -180 ry 0 rz 90 deg; joints [6.346, -25.657, 98.075, 190.891, 21.6, -185.204]
  MoveL 219 to (-189, -173.6, 20) mm, rotated rx -180 ry 0 rz 90 deg; joints [6.346, -26.631, 98.622, 191.1, 21.18, -185.427]
  Set speed (1000.0 mm/s)
  MoveL 220 to (-189, -218.31, 20) mm, rotated rx 180 ry 0 rz 90 deg; joints [6.184, -25.975, 96.038, 191.847, 19.282, -186.387]
  Set speed (50.0 mm/s)
  MoveL 221 to (-189, -218.31, 0) mm, rotated rx -180 ry 0 rz 90 deg; joints [6.184, -25.017, 95.495, 191.609, 19.688, -186.134]
  MoveL 222 to (-189, -218.31, 20) mm, rotated rx 180 ry 0 rz 90 deg; joints [6.184, -25.975, 96.038, 191.847, 19.282, -186.387]
  Set speed (1000.0 mm/s)
  MoveL 223 to (-189, -263.02, 20) mm, rotated rx 180 ry 0 rz 90 deg; joints [6.031, -25.251, 93.388, 192.782, 17.388, -187.522]
  Set speed (50.0 mm/s)
  MoveL 224 to (-189, -263.02, 0) mm, rotated rx -180 ry 0 rz 90 deg; joints [6.031, -24.309, 92.848, 192.505, 17.78, -187.231]
  MoveL 225 to (-189, -263.02, 20) mm, rotated rx 180 ry 0 rz 90 deg; joints [6.031, -25.251, 93.388, 192.782, 17.388, -187.522]
  Set speed (1000.0 mm/s)
  MoveL 226 to (-189, -307.73, 20) mm, rotated rx 180 ry 0 rz 90 deg; joints [5.885, -24.459, 90.667, 193.974, 15.497, -188.906]
  Set speed (50.0 mm/s)
  MoveL 227 to (-189, -307.73, 0) mm, rotated rx -180 ry 0 rz 90 deg; joints [5.885, -23.532, 90.129, 193.644, 15.874, -188.563]
  MoveL 228 to (-189, -307.73, 20) mm, rotated rx 180 ry 0 rz 90 deg; joints [5.885, -24.459, 90.667, 193.974, 15.497, -188.906]
  Set speed (1000.0 mm/s)
  MoveL 229 to (-189, -352.44, 20) mm, rotated rx 180 ry 0 rz 90 deg; joints [5.746, -23.6, 87.869, 195.534, 13.607, -190.647]
  Set speed (50.0 mm/s)
  MoveL 230 to (-189, -352.44, 0) mm, rotated rx 180 ry 0 rz 90 deg; joints [5.746, -22.687, 87.331, 195.129, 13.969, -190.23]
  MoveL 231 to (-189, -352.44, 20) mm, rotated rx 180 ry 0 rz 90 deg; joints [5.746, -23.6, 87.869, 195.534, 13.607, -190.647]
  Set speed (1000.0 mm/s)
  MoveL 232 to (-189, -397.15, 20) mm, rotated rx 180 ry 0 rz 90 deg; joints [5.613, -22.672, 84.987, 197.643, 11.718, -192.93]
  Set speed (50.0 mm/s)
  MoveL 233 to (-189, -397.15, 0) mm, rotated rx 180 ry 0 rz 90 deg; joints [5.613, -21.771, 84.448, 197.13, 12.063, -192.405]
  MoveL 234 to (-189, -397.15, 20) mm, rotated rx 180 ry 0 rz 90 deg; joints [5.613, -22.672, 84.987, 197.643, 11.718, -192.93]
  Set speed (1000.0 mm/s)
  MoveL 235 to (-189, -441.86, 20) mm, rotated rx -180 ry 0 rz 90 deg; joints [5.486, -21.672, 82.015, 200.628, 9.833, -196.082]
  Set speed (50.0 mm/s)
  MoveL 236 to (-189, -441.86, 0) mm, rotated rx -180 ry 0 rz 90 deg; joints [5.486, -20.783, 81.473, 199.945, 10.159, -195.387]
  MoveL 237 to (-189, -441.86, 20) mm, rotated rx -180 ry 0 rz 90 deg; joints [5.486, -21.672, 82.015, 200.628, 9.833, -196.082]
  Set speed (1000.0 mm/s)
  MoveL 238 to (-189, -486.57, 20) mm, rotated rx -180 ry 0 rz 90 deg; joints [5.365, -20.598, 78.942, 205.124, 7.966, -200.737]
  Set speed (50.0 mm/s)
  MoveL 239 to (-189, -486.57, 0) mm, rotated rx 180 ry 0 rz 90 deg; joints [5.365, -19.719, 78.396, 204.15, 8.269, -199.752]
  MoveL 240 to (-189, -486.57, 20) mm, rotated rx -180 ry 0 rz 90 deg; joints [5.365, -20.598, 78.942, 205.124, 7.966, -200.737]
  Set speed (1000.0 mm/s)
  MoveL 241 to (-189, -531.28, 20) mm, rotated rx -180 ry 0 rz 90 deg; joints [5.249, -19.445, 75.757, 212.494, 6.152, -208.26]
  Set speed (50.0 mm/s)
  MoveL 242 to (-189, -531.28, 0) mm, rotated rx 180 ry 0 rz 90 deg; joints [5.249, -18.575, 75.206, 210.974, 6.423, -206.731]
  MoveL 243 to (-189, -531.28, 20) mm, rotated rx -180 ry 0 rz 90 deg; joints [5.249, -19.445, 75.757, 212.494, 6.152, -208.26]
  Set speed (1000.0 mm/s)
  MoveL 244 to (-189, -575.99, 20) mm, rotated rx -180 ry 0 rz 90 deg; joints [5.138, -18.208, 72.448, 225.975, 4.496, -221.889]
  Set speed (50.0 mm/s)
  MoveL 245 to (-189, -575.99, 0) mm, rotated rx 180 ry 0 rz 90 deg; joints [5.138, -17.345, 71.889, 223.33, 4.711, -219.236]
  MoveL 246 to (-189, -575.99, 20) mm, rotated rx -180 ry 0 rz 90 deg; joints [5.138, -18.208, 72.448, 225.975, 4.496, -221.889]
  Set speed (1000.0 mm/s)
  MoveL 247 to (-0.17, -575.99, 20) mm, rotated rx 180 ry 0 rz 90 deg; joints [0.005, -18.45, 73.089, 180.046, 3.639, -180.042]
  Set speed (50.0 mm/s)
  MoveL 248 to (-0.17, -575.99, 0) mm, rotated rx 180 ry 0 rz 90 deg; joints [0.005, -17.586, 72.531, 180.042, 3.945, -180.039]
  MoveL 249 to (-0.17, -575.99, 20) mm, rotated rx -180 ry 0 rz 90 deg; joints [0.005, -18.45, 73.089, 180.046, 3.639, -180.042]
  Set speed (1000.0 mm/s)
  MoveL 250 to (-0.17, -531.37, 20) mm, rotated rx 180 ry 0 rz 90 deg; joints [0.005, -19.673, 76.38, 180.03, 5.707, -180.026]
  Set speed (50.0 mm/s)
  MoveL 251 to (-0.17, -531.37, 0) mm, rotated rx 180 ry 0 rz 90 deg; joints [0.005, -18.802, 75.83, 180.028, 6.028, -180.025]
  MoveL 252 to (-0.17, -531.37, 20) mm, rotated rx 180 ry 0 rz 90 deg; joints [0.005, -19.673, 76.38, 180.03, 5.707, -180.026]
  Set speed (1000.0 mm/s)
  MoveL 253 to (-0.17, -486.76, 20) mm, rotated rx -180 ry 0 rz 90 deg; joints [0.005, -20.813, 79.548, 180.023, 7.735, -180.019]
  Set speed (50.0 mm/s)
  MoveL 254 to (-0.17, -486.76, 0) mm, rotated rx -180 ry 0 rz 90 deg; joints [0.005, -19.932, 79.004, 180.022, 8.072, -180.018]
  MoveL 255 to (-0.17, -486.76, 20) mm, rotated rx -180 ry 0 rz 90 deg; joints [0.005, -20.813, 79.548, 180.023, 7.735, -180.019]
  Set speed (1000.0 mm/s)
  MoveL 256 to (-0.17, -442.14, 20) mm, rotated rx -180 ry 0 rz 90 deg; joints [0.005, -21.875, 82.608, 180.018, 9.733, -180.014]
  Set speed (50.0 mm/s)
  MoveL 257 to (-0.17, -442.14, 0) mm, rotated rx 180 ry 0 rz 90 deg; joints [0.005, -20.984, 82.068, 180.018, 10.084, -180.014]
  MoveL 258 to (-0.17, -442.14, 20) mm, rotated rx -180 ry 0 rz 90 deg; joints [0.005, -21.875, 82.608, 180.018, 9.733, -180.014]
  Set speed (1000.0 mm/s)
  MoveL 259 to (163, -380.99, 20) mm, rotated rx -180 ry 0 rz 90 deg; joints [-4.886, -23.066, 86.194, 165.554, 12.407, -169.679]
  Set speed (50.0 mm/s)
  MoveL 260 to (163, -380.99, 0) mm, rotated rx -180 ry 0 rz 90 deg; joints [-4.886, -22.16, 85.656, 165.959, 12.763, -170.093]
  MoveL 261 to (163, -380.99, 20) mm, rotated rx -180 ry 0 rz 90 deg; joints [-4.886, -23.066, 86.194, 165.554, 12.407, -169.679]
  Set speed (1000.0 mm/s)
  MoveL 262 to (116.33, -380.99, 20) mm, rotated rx 180 ry 0 rz 90 deg; joints [-3.491, -23.137, 86.415, 169.736, 12.419, -172.685]
  Set speed (50.0 mm/s)
  MoveL 263 to (116.33, -380.99, 0) mm, rotated rx 180 ry 0 rz 90 deg; joints [-3.491, -22.231, 85.877, 170.025, 12.781, -172.982]
  MoveL 264 to (116.33, -380.99, 20) mm, rotated rx 180 ry 0 rz 90 deg; joints [-3.491, -23.137, 86.415, 169.736, 12.419, -172.685]
  Set speed (1000.0 mm/s)
  MoveL 265 to (69.67, -380.99, 20) mm, rotated rx -180 ry 0 rz 90 deg; joints [-2.092, -23.185, 86.562, 173.871, 12.428, -175.64]
  Set speed (50.0 mm/s)
  MoveL 266 to (69.67, -380.99, 0) mm, rotated rx 180 ry 0 rz 90 deg; joints [-2.092, -22.277, 86.024, 174.045, 12.795, -175.818]
  MoveL 267 to (69.67, -380.99, 20) mm, rotated rx -180 ry 0 rz 90 deg; joints [-2.092, -23.185, 86.562, 173.871, 12.428, -175.64]
  Set speed (1000.0 mm/s)
  MoveL 268 to (23, -380.99, 20) mm, rotated rx 180 ry 0 rz 90 deg; joints [-0.691, -23.208, 86.636, 177.98, 12.433, -178.564]
  Set speed (50.0 mm/s)
  MoveL 269 to (23, -380.99, 0) mm, rotated rx 180 ry 0 rz 90 deg; joints [-0.691, -22.301, 86.097, 178.037, 12.802, -178.623]
  MoveL 270 to (23, -380.99, 20) mm, rotated rx 180 ry 0 rz 90 deg; joints [-0.691, -23.208, 86.636, 177.98, 12.433, -178.564]
  Set speed (1000.0 mm/s)
  MoveL 271 to (-0.17, -397.53, 20) mm, rotated rx 180 ry 0 rz 90 deg; joints [0.005, -22.863, 85.57, 180.016, 11.707, -180.011]
  Set speed (50.0 mm/s)
  MoveL 272 to (-0.17, -397.53, 0) mm, rotated rx -180 ry 0 rz 90 deg; joints [0.005, -21.96, 85.031, 180.015, 12.071, -180.011]
  MoveL 273 to (-0.17, -397.53, 20) mm, rotated rx 180 ry 0 rz 90 deg; joints [0.005, -22.863, 85.57, 180.016, 11.707, -180.011]
  Set speed (1000.0 mm/s)
  MoveL 274 to (-23, -380.99, 20) mm, rotated rx -180 ry 0 rz 90 deg; joints [0.691, -23.208, 86.636, 182.02, 12.433, -181.436]
  Set speed (50.0 mm/s)
  MoveL 275 to (-23, -380.99, 0) mm, rotated rx -180 ry 0 rz 90 deg; joints [0.691, -22.301, 86.097, 181.963, 12.802, -181.377]
  MoveL 276 to (-23, -380.99, 20) mm, rotated rx -180 ry 0 rz 90 deg; joints [0.691, -23.208, 86.636, 182.02, 12.433, -181.436]
  Set speed (1000.0 mm/s)
  MoveL 277 to (-69.67, -380.99, 20) mm, rotated rx 180 ry 0 rz 90 deg; joints [2.092, -23.185, 86.562, 186.129, 12.428, -184.36]
  Set speed (50.0 mm/s)
  MoveL 278 to (-69.67, -380.99, 0) mm, rotated rx -180 ry 0 rz 90 deg; joints [2.092, -22.277, 86.024, 185.955, 12.795, -184.182]
  MoveL 279 to (-69.67, -380.99, 20) mm, rotated rx 180 ry 0 rz 90 deg; joints [2.092, -23.185, 86.562, 186.129, 12.428, -184.36]
  Set speed (1000.0 mm/s)
  MoveL 280 to (-116.33, -380.99, 20) mm, rotated rx -180 ry 0 rz 90 deg; joints [3.491, -23.137, 86.415, 190.264, 12.419, -187.315]
  Set speed (50.0 mm/s)
  MoveL 281 to (-116.33, -380.99, 0) mm, rotated rx 180 ry 0 rz 90 deg; joints [3.491, -22.231, 85.877, 189.975, 12.781, -187.018]
  MoveL 282 to (-116.33, -380.99, 20) mm, rotated rx -180 ry 0 rz 90 deg; joints [3.491, -23.137, 86.415, 190.264, 12.419, -187.315]
  Set speed (1000.0 mm/s)
  MoveL 283 to (-163, -380.99, 20) mm, rotated rx 180 ry 0 rz 90 deg; joints [4.886, -23.066, 86.194, 194.446, 12.407, -190.321]
  Set speed (50.0 mm/s)
  MoveL 284 to (-163, -380.99, 0) mm, rotated rx 180 ry 0 rz 90 deg; joints [4.886, -22.16, 85.656, 194.041, 12.763, -189.907]
  MoveL 285 to (-163, -380.99, 20) mm, rotated rx 180 ry 0 rz 90 deg; joints [4.886, -23.066, 86.194, 194.446, 12.407, -190.321]
  Set speed (1000.0 mm/s)
  MoveL 286 to (-0.17, -352.91, 20) mm, rotated rx -180 ry 0 rz 90 deg; joints [0.005, -23.78, 88.442, 180.014, 13.662, -180.009]
  Set speed (50.0 mm/s)
  MoveL 287 to (-0.17, -352.91, 0) mm, rotated rx 180 ry 0 rz 90 deg; joints [0.005, -22.864, 87.904, 180.013, 14.04, -180.009]
  MoveL 288 to (-0.17, -352.91, 20) mm, rotated rx -180 ry 0 rz 90 deg; joints [0.005, -23.78, 88.442, 180.014, 13.662, -180.009]
  Set speed (1000.0 mm/s)
  MoveL 289 to (-0.17, -308.3, 20) mm, rotated rx 180 ry 0 rz 90 deg; joints [0.005, -24.628, 91.233, 180.012, 15.605, -180.008]
  Set speed (50.0 mm/s)
  MoveL 290 to (-0.17, -308.3, 0) mm, rotated rx 180 ry 0 rz 90 deg; joints [0.005, -23.698, 90.694, 180.012, 15.996, -180.008]
  MoveL 291 to (-0.17, -308.3, 20) mm, rotated rx 180 ry 0 rz 90 deg; joints [0.005, -24.628, 91.233, 180.012, 15.605, -180.008]
  Set speed (1000.0 mm/s)
  MoveL 292 to (-0.17, -263.68, 20) mm, rotated rx 180 ry 0 rz 90 deg; joints [0.005, -25.408, 93.948, 180.011, 17.541, -180.007]
  Set speed (50.0 mm/s)
  MoveL 293 to (-0.17, -263.68, 0) mm, rotated rx 180 ry 0 rz 90 deg; joints [0.005, -24.463, 93.408, 180.011, 17.945, -180.006]
  MoveL 294 to (-0.17, -263.68, 20) mm, rotated rx 180 ry 0 rz 90 deg; joints [0.005, -25.408, 93.948, 180.011, 17.541, -180.007]
  Set speed (1000.0 mm/s)
  MoveL 295 to (-0.17, -219.07, 20) mm, rotated rx -180 ry 0 rz 90 deg; joints [0.006, -26.12, 96.593, 180.011, 19.473, -180.006]
  Set speed (50.0 mm/s)
  MoveL 296 to (-0.17, -219.07, 0) mm, rotated rx -180 ry 0 rz 90 deg; joints [0.006, -25.159, 96.049, 180.01, 19.891, -180.005]
  MoveL 297 to (-0.17, -219.07, 20) mm, rotated rx -180 ry 0 rz 90 deg; joints [0.006, -26.12, 96.593, 180.011, 19.473, -180.006]
  Set speed (1000.0 mm/s)
  MoveL 298 to (-0.17, -174.45, 20) mm, rotated rx -180 ry 0 rz 90 deg; joints [0.006, -26.765, 99.173, 180.01, 21.408, -180.005]
  Set speed (50.0 mm/s)
  MoveL 299 to (-0.17, -174.45, 0) mm, rotated rx 180 ry 0 rz 90 deg; joints [0.006, -25.786, 98.625, 180.01, 21.838, -180.005]
  MoveL 300 to (-0.17, -174.45, 20) mm, rotated rx -180 ry 0 rz 90 deg; joints [0.006, -26.765, 99.173, 180.01, 21.408, -180.005]
  Set speed (1000.0 mm/s)
  MoveL 301 to (-0.17, -129.84, 20) mm, rotated rx 180 ry 0 rz 90 deg; joints [0.006, -27.341, 101.69, 180.009, 23.349, -180.004]
  Set speed (50.0 mm/s)
  MoveL 302 to (-0.17, -129.84, 0) mm, rotated rx -180 ry 0 rz 90 deg; joints [0.006, -26.345, 101.137, 180.009, 23.792, -180.004]
  MoveL 303 to (-0.17, -129.84, 20) mm, rotated rx 180 ry 0 rz 90 deg; joints [0.006, -27.341, 101.69, 180.009, 23.349, -180.004]
  Set speed (1000.0 mm/s)
  MoveL 304 to (-0.17, -85.22, 20) mm, rotated rx 180 ry 0 rz 90 deg; joints [0.006, -27.847, 104.149, 180.009, 25.302, -180.003]
  Set speed (50.0 mm/s)
  MoveL 305 to (-0.17, -85.22, 0) mm, rotated rx -180 ry 0 rz 90 deg; joints [0.006, -26.832, 103.59, 180.009, 25.757, -180.003]
  MoveL 306 to (-0.17, -85.22, 20) mm, rotated rx 180 ry 0 rz 90 deg; joints [0.006, -27.847, 104.149, 180.009, 25.302, -180.003]
  Set speed (1000.0 mm/s)
  MoveL 307 to (-0.17, -40.61, 20) mm, rotated rx 180 ry 0 rz 90 deg; joints [0.006, -28.281, 106.551, 180.009, 27.27, -180.003]
  Set speed (50.0 mm/s)
  MoveL 308 to (-0.17, -40.61, 0) mm, rotated rx -180 ry 0 rz 90 deg; joints [0.006, -27.247, 105.984, 180.008, 27.738, -180.003]
  MoveL 309 to (-0.17, -40.61, 20) mm, rotated rx 180 ry 0 rz 90 deg; joints [0.006, -28.281, 106.551, 180.009, 27.27, -180.003]
  Set speed (1000.0 mm/s)
  MoveL 310 to (-0.17, 4.01, 20) mm, rotated rx -180 ry 0 rz 90 deg; joints [0.006, -28.642, 108.899, 180.008, 29.258, -180.002]
  Set speed (50.0 mm/s)
  MoveL 311 to (-0.17, 4.01, 0) mm, rotated rx -180 ry 0 rz 90 deg; joints [0.006, -27.587, 108.325, 180.008, 29.738, -180.002]
  MoveL 312 to (-0.17, 4.01, 20) mm, rotated rx -180 ry 0 rz 90 deg; joints [0.006, -28.642, 108.899, 180.008, 29.258, -180.002]
  Set speed (1000.0 mm/s)
  MoveL 313 to (-0.17, 48.63, 20) mm, rotated rx -180 ry 0 rz 90 deg; joints [0.007, -28.925, 111.195, 180.008, 31.27, -180.002]
  Set speed (50.0 mm/s)
  MoveL 314 to (-0.17, 48.63, 0) mm, rotated rx -180 ry 0 rz 90 deg; joints [0.007, -27.849, 110.611, 180.008, 31.763, -180.002]
  MoveL 315 to (-0.17, 48.63, 20) mm, rotated rx -180 ry 0 rz 90 deg; joints [0.007, -28.925, 111.195, 180.008, 31.27, -180.002]
  Set speed (1000.0 mm/s)
  MoveL 316 to (-0.17, 93.24, 20) mm, rotated rx 180 ry 0 rz 90 deg; joints [0.007, -29.127, 113.439, 180.008, 33.312, -180.001]
  Set speed (50.0 mm/s)
  MoveL 317 to (-0.17, 93.24, 0) mm, rotated rx 180 ry 0 rz 90 deg; joints [0.007, -28.029, 112.845, 180.008, 33.817, -180.001]
  MoveL 318 to (-0.17, 93.24, 20) mm, rotated rx 180 ry 0 rz 90 deg; joints [0.007, -29.127, 113.439, 180.008, 33.312, -180.001]
  Set speed (1000.0 mm/s)
  MoveL 319 to (-0.17, 137.86, 20) mm, rotated rx -180 ry 0 rz 90 deg; joints [0.007, -29.244, 115.633, 180.008, 35.39, -180.001]
  Set speed (50.0 mm/s)
  MoveL 320 to (-0.17, 137.86, 0) mm, rotated rx -180 ry 0 rz 90 deg; joints [0.007, -28.123, 115.028, 180.008, 35.905, -180.001]
  MoveL 321 to (-0.17, 137.86, 20) mm, rotated rx -180 ry 0 rz 90 deg; joints [0.007, -29.244, 115.633, 180.008, 35.39, -180.001]
  Set speed (1000.0 mm/s)
  MoveL 322 to (163, 179.01, 20) mm, rotated rx 180 ry 0 rz 90 deg; joints [-6.9, -29.272, 117.143, 172.764, 36.887, -179.574]
  Set speed (50.0 mm/s)
  MoveL 323 to (163, 179.01, 0) mm, rotated rx 180 ry 0 rz 90 deg; joints [-6.9, -28.135, 116.529, 172.85, 37.406, -179.682]
  MoveL 324 to (163, 179.01, 20) mm, rotated rx 180 ry 0 rz 90 deg; joints [-6.9, -29.272, 117.143, 172.764, 36.887, -179.574]
  Set speed (1000.0 mm/s)
  MoveL 325 to (116.33, 179.01, 20) mm, rotated rx -180 ry 0 rz 90 deg; joints [-4.936, -29.272, 117.373, 174.851, 37.108, -179.729]
  Set speed (50.0 mm/s)
  MoveL 326 to (116.33, 179.01, 0) mm, rotated rx 180 ry 0 rz 90 deg; joints [-4.936, -28.133, 116.758, 174.912, 37.63, -179.806]
  MoveL 327 to (116.33, 179.01, 20) mm, rotated rx -180 ry 0 rz 90 deg; joints [-4.936, -29.272, 117.373, 174.851, 37.108, -179.729]
  Set speed (1000.0 mm/s)
  MoveL 328 to (69.67, 179.01, 20) mm, rotated rx -180 ry 0 rz 90 deg; joints [-2.961, -29.272, 117.526, 176.922, 37.257, -179.851]
  Set speed (50.0 mm/s)
  MoveL 329 to (69.67, 179.01, 0) mm, rotated rx 180 ry 0 rz 90 deg; joints [-2.961, -28.13, 116.91, 176.958, 37.781, -179.897]
  MoveL 330 to (69.67, 179.01, 20) mm, rotated rx -180 ry 0 rz 90 deg; joints [-2.961, -29.272, 117.526, 176.922, 37.257, -179.851]
  Set speed (1000.0 mm/s)
  MoveL 331 to (23, 179.01, 20) mm, rotated rx 180 ry 0 rz 90 deg; joints [-0.978, -29.271, 117.602, 178.985, 37.331, -179.953]
  Set speed (50.0 mm/s)
  MoveL 332 to (23, 179.01, 0) mm, rotated rx 180 ry 0 rz 90 deg; joints [-0.978, -28.129, 116.986, 178.997, 37.857, -179.968]
  MoveL 333 to (23, 179.01, 20) mm, rotated rx 180 ry 0 rz 90 deg; joints [-0.978, -29.271, 117.602, 178.985, 37.331, -179.953]
  Set speed (1000.0 mm/s)
  MoveL 334 to (-0.17, 182.47, 20) mm, rotated rx 180 ry 0 rz 90 deg; joints [0.007, -29.27, 117.776, 180.007, 37.506, -180]
  Set speed (50.0 mm/s)
  MoveL 335 to (-0.17, 182.47, 0) mm, rotated rx -180 ry 0 rz 90 deg; joints [0.007, -28.126, 117.158, 180.007, 38.032, -180]
  MoveL 336 to (-0.17, 182.47, 20) mm, rotated rx 180 ry 0 rz 90 deg; joints [0.007, -29.27, 117.776, 180.007, 37.506, -180]
  Set speed (1000.0 mm/s)
  MoveL 337 to (-23, 179.01, 20) mm, rotated rx -180 ry 0 rz 90 deg; joints [0.978, -29.271, 117.602, 181.015, 37.331, -180.047]
  Set speed (50.0 mm/s)
  MoveL 338 to (-23, 179.01, 0) mm, rotated rx -180 ry 0 rz 90 deg; joints [0.978, -28.129, 116.986, 181.003, 37.857, -180.032]
  MoveL 339 to (-23, 179.01, 20) mm, rotated rx -180 ry 0 rz 90 deg; joints [0.978, -29.271, 117.602, 181.015, 37.331, -180.047]
  Set speed (1000.0 mm/s)
  MoveL 340 to (-69.67, 179.01, 20) mm, rotated rx -180 ry 0 rz 90 deg; joints [2.961, -29.272, 117.526, 183.078, 37.257, -180.149]
  Set speed (50.0 mm/s)
  MoveL 341 to (-69.67, 179.01, 0) mm, rotated rx -180 ry 0 rz 90 deg; joints [2.961, -28.13, 116.91, 183.042, 37.781, -180.103]
  MoveL 342 to (-69.67, 179.01, 20) mm, rotated rx -180 ry 0 rz 90 deg; joints [2.961, -29.272, 117.526, 183.078, 37.257, -180.149]
  Set speed (1000.0 mm/s)
  MoveL 343 to (-116.33, 179.01, 20) mm, rotated rx -180 ry 0 rz 90 deg; joints [4.936, -29.272, 117.373, 185.149, 37.108, -180.271]
  Set speed (50.0 mm/s)
  MoveL 344 to (-116.33, 179.01, 0) mm, rotated rx -180 ry 0 rz 90 deg; joints [4.936, -28.133, 116.758, 185.088, 37.63, -180.194]
  MoveL 345 to (-116.33, 179.01, 20) mm, rotated rx -180 ry 0 rz 90 deg; joints [4.936, -29.272, 117.373, 185.149, 37.108, -180.271]
  Set speed (1000.0 mm/s)
  MoveL 346 to (-163, 179.01, 20) mm, rotated rx 180 ry 0 rz 90 deg; joints [6.9, -29.272, 117.143, 187.236, 36.887, -180.426]
  Set speed (50.0 mm/s)
  MoveL 347 to (-163, 179.01, 0) mm, rotated rx -180 ry 0 rz 90 deg; joints [6.9, -28.135, 116.529, 187.15, 37.406, -180.318]
  MoveL 348 to (-163, 179.01, 20) mm, rotated rx 180 ry 0 rz 90 deg; joints [6.9, -29.272, 117.143, 187.236, 36.887, -180.426]
  Set speed (1000.0 mm/s)
  MoveL 349 to (-0.17, 227.09, 20) mm, rotated rx 180 ry 0 rz 90 deg; joints [0.007, -29.2, 119.869, 180.007, 39.669, -180]
  Set speed (50.0 mm/s)
  MoveL 350 to (-0.17, 227.09, 0) mm, rotated rx 180 ry 0 rz 90 deg; joints [0.007, -28.033, 119.238, 180.007, 40.205, -180]
  MoveL 351 to (-0.17, 227.09, 20) mm, rotated rx 180 ry 0 rz 90 deg; joints [0.007, -29.2, 119.869, 180.007, 39.669, -180]
  Set speed (1000.0 mm/s)
  MoveL 352 to (-0.17, 271.7, 20) mm, rotated rx -180 ry 0 rz 90 deg; joints [0.008, -29.028, 121.911, 180.007, 41.883, -179.999]
  Set speed (50.0 mm/s)
  MoveL 353 to (-0.17, 271.7, 0) mm, rotated rx 180 ry 0 rz 90 deg; joints [0.008, -27.837, 121.265, 180.007, 42.428, -179.999]
  MoveL 354 to (-0.17, 271.7, 20) mm, rotated rx -180 ry 0 rz 90 deg; joints [0.008, -29.028, 121.911, 180.007, 41.883, -179.999]
  Set speed (1000.0 mm/s)
  MoveL 355 to (-0.17, 316.32, 20) mm, rotated rx -180 ry 0 rz 90 deg; joints [0.008, -28.746, 123.901, 180.007, 44.155, -179.999]
  Set speed (50.0 mm/s)
  MoveL 356 to (-0.17, 316.32, 0) mm, rotated rx 180 ry 0 rz 90 deg; joints [0.008, -27.532, 123.24, 180.007, 44.708, -179.999]
  MoveL 357 to (-0.17, 316.32, 20) mm, rotated rx -180 ry 0 rz 90 deg; joints [0.008, -28.746, 123.901, 180.007, 44.155, -179.999]
  Set speed (1000.0 mm/s)
  MoveL 358 to (-0.17, 360.93, 20) mm, rotated rx -180 ry 0 rz 90 deg; joints [0.008, -28.346, 125.837, 180.007, 46.491, -179.998]
  Set speed (50.0 mm/s)
  MoveL 359 to (-0.17, 360.93, 0) mm, rotated rx 180 ry 0 rz 90 deg; joints [0.008, -27.109, 125.159, 180.007, 47.051, -179.998]
  MoveL 360 to (-0.17, 360.93, 20) mm, rotated rx -180 ry 0 rz 90 deg; joints [0.008, -28.346, 125.837, 180.007, 46.491, -179.998]
  Set speed (1000.0 mm/s)
  MoveL 361 to (-0.17, 405.55, 20) mm, rotated rx -180 ry 0 rz 90 deg; joints [0.009, -27.819, 127.719, 180.007, 48.9, -179.998]
  Set speed (50.0 mm/s)
  MoveL 362 to (-0.17, 405.55, 0) mm, rotated rx 180 ry 0 rz 90 deg; joints [0.009, -26.56, 127.023, 180.007, 49.463, -179.998]
  MoveL 363 to (-0.17, 405.55, 20) mm, rotated rx -180 ry 0 rz 90 deg; joints [0.009, -27.819, 127.719, 180.007, 48.9, -179.998]
  MoveL 364 to (-0.17, 405.55, 20) mm, rotated rx -180 ry 0 rz 90 deg; joints [0.009, -27.819, 127.719, 180.007, 48.9, -179.998]
  Set speed (1000.0 mm/s)
  MoveL 365 to (-0.17, 405.55, 20) mm, rotated rx -180 ry 0 rz 90 deg; joints [0.009, -27.819, 127.719, 180.007, 48.9, -179.998]
  MoveL 366 to (-0.17, 405.55, 120) mm, rotated rx 180 ry 0 rz 90 deg; joints [0.009, -34.349, 130.969, 180.008, 45.62, -179.999]
